TYPE SocketConnect :
(
	SocketInit:=0,
	SocketConnect,
	SocketSend,
	SocketRecive,
	SocketClose,
	SocketReset
)INT;
END_TYPE

(* stored: Version 1.1.0.1, ProductVersion 3.1.4022.16
   DUT SocketConnect: Id {e7cf9d18-caf8-405c-bac1-8bed08dc72e8} *)
